FUNCTION_BLOCK FB_StateMachine
VAR_INPUT
END_VAR
VAR_OUTPUT
END_VAR
VAR
	fbMotionSelector : FB_MotionRefSelector;
	fbThetaBoom : FB_ThetaBoom;
END_VAR

IF (G_ControllerGreenCrane.bEnable) THEN
	G_ControllerGreenCrane.eStatus := E_Status.Ready;
	IF (G_ControllerGreenCrane.bMode) THEN
		G_ControllerGreenCrane.eMode := E_Mode.Auto;
		IF (G_ControllerGreenCrane.bStartAutoMode) THEN
			G_ControllerGreenCrane.bLamp := TRUE;
			G_ControllerGreenCrane.bStart := FALSE;
		ELSE
			G_ControllerGreenCrane.bLamp := G_ControllerGreenCrane.bStart := FALSE;
		END_IF
	ELSE  
		G_ControllerGreenCrane.eMode := E_Mode.Manual;
		G_ControllerGreenCrane.bLamp := G_ControllerGreenCrane.bStart;
		IF (G_ControllerGreenCrane.bStart) THEN
			G_ControllerGreenCrane.eStatus := E_Status.Running;
		END_IF		
	END_IF
ELSE
	G_ControllerGreenCrane.bStart := G_ControllerGreenCrane.bLamp := FALSE;
	G_ControllerGreenCrane.eStatus := E_Status.NotReady;
	IF (G_ControllerGreenCrane.bMode) THEN
		G_ControllerGreenCrane.eMode := E_Mode.Auto;
	ELSE  
		G_ControllerGreenCrane.eMode := E_Mode.Manual;
	END_IF
END_IF

IF (G_ControllerGreenCrane.bLamp) THEN
	G_ControllerGreenCrane.fTimer := G_ControllerGreenCrane.fTimer + 0.01;
ELSE 
	G_ControllerGreenCrane.fTimer := 0.0;
END_IF


fbMotionSelector(Auto1Man0 := G_ControllerGreenCrane.bMode, xCylRefGenm := 0, vCylRefGenm := 0, vCylJoyms := G_ControllerGreenCrane.fVelRef);
fbThetaBoom(xCylm := G_CylinderState.xm, thetaBoom => G_CylinderState.thetaBoom);

END_FUNCTION_BLOCK

(* stored: Version 1.1.0.1, ProductVersion 3.1.4024.12
   POU FB_StateMachine: Id {1198fdea-b4e3-4647-9eef-33003000b939}, SpecialFunc None *)
